FUNCTION MODULO : LREAL
VAR_INPUT
	fValue : LREAL;
	fDenom : LREAL := 360;
END_VAR
VAR
END_VAR

MODULO := fValue - (TRUNC(fValue / fDenom) * fDenom);

END_FUNCTION

(* stored: Version 1.1.0.1, ProductVersion 3.1.4022.10
   POU MODULO: Id {a405c42f-68fb-47d3-879d-de49f61e9ee1}, SpecialFunc None *)
